{attribute 'qualified_only'}
VAR_GLOBAL
	B1 :BOOL; 	// Druckschalter
	B2 :BOOL;   // Temperaturfühler Kompressor
	F1 :BOOL;   // Störung Motorschutzschalter
	S1 :BOOL;   // Taster Aus
	S2 :BOOL;   // Taster Ein
END_VAR

(* stored: Version 1.1.0.1, ProductVersion 3.1.4024.5
   GVL SimDI: Id {c2d05302-d374-4f85-80dd-41006a3e3277} *)
